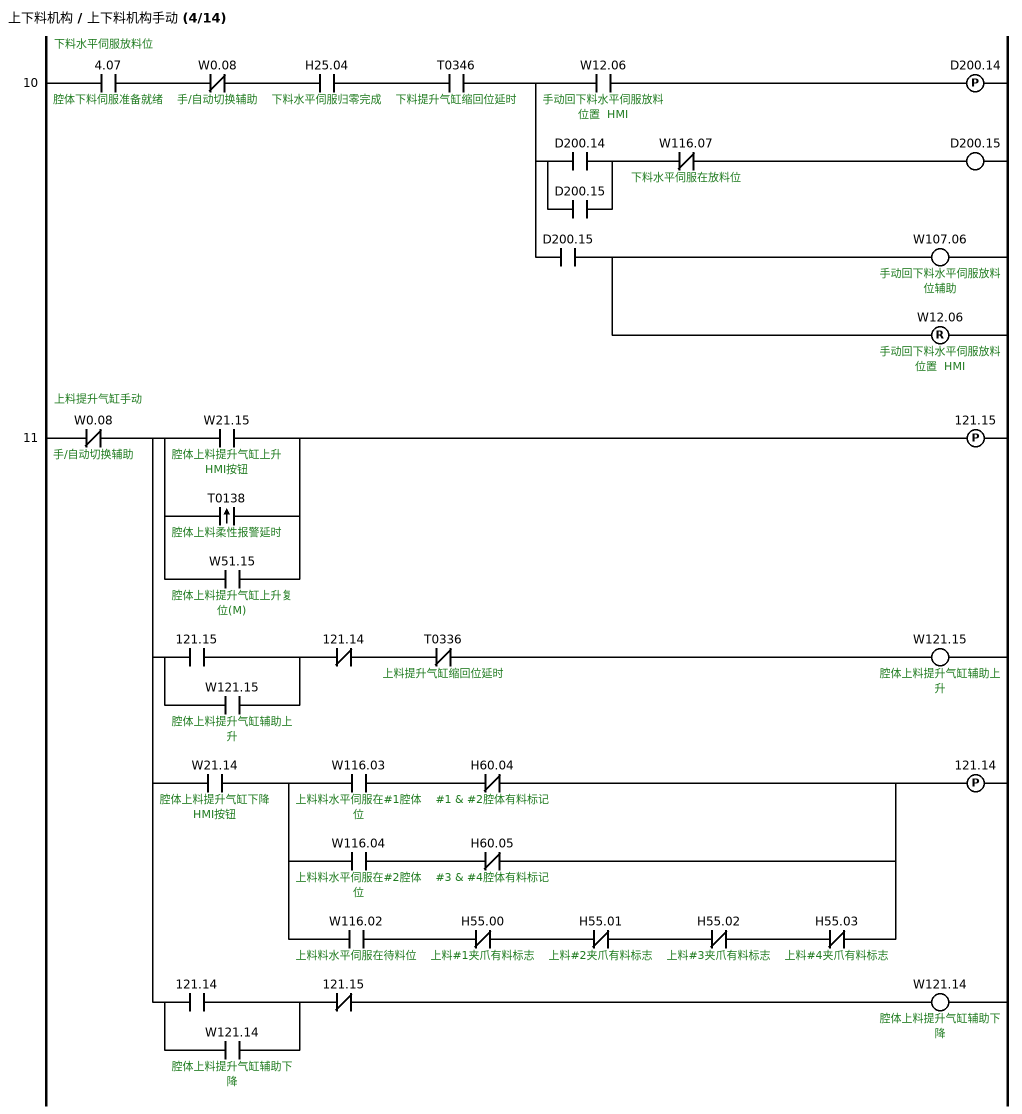
; [picture p192: 上下料机构 / 上下料机构手动, rungs 10-11]
; rung 10: 下料水平伺服放料位
LD 4.07  ; 腔体下料伺服准备就绪
ANDNOT W0.08  ; 手/自动切换辅助
AND H25.04  ; 下料水平伺服归零完成
AND T0346  ; 下料提升气缸缩回位延时
OUT TR0
AND W12.06  ; 手动回下料水平伺服放料位置  HMI
DIFU(013) D200.14
LD TR0
LD D200.14
OR D200.15
ANDLD
ANDNOT W116.07  ; 下料水平伺服在放料位
OUT D200.15
LD TR0
AND D200.15
OUT W107.06  ; 手动回下料水平伺服放料位辅助
RSET W12.06  ; 手动回下料水平伺服放料位置  HMI
; rung 11: 上料提升气缸手动
LDNOT W0.08  ; 手/自动切换辅助
OUT TR0
LD W21.15  ; 腔体上料提升气缸上升   HMI按钮
@OR T0138  ; 腔体上料柔性报警延时
OR W51.15  ; 腔体上料提升气缸上升复位(M)
ANDLD
DIFU(013) 121.15
LD TR0
LD 121.15
OR W121.15  ; 腔体上料提升气缸辅助上升
ANDLD
ANDNOT 121.14
ANDNOT T0336  ; 上料提升气缸缩回位延时
OUT W121.15  ; 腔体上料提升气缸辅助上升
LD TR0
AND W21.14  ; 腔体上料提升气缸下降   HMI按钮
LD W116.03  ; 上料料水平伺服在#1腔体位
ANDNOT H60.04  ; #1 & #2腔体有料标记
LD W116.04  ; 上料料水平伺服在#2腔体位
ANDNOT H60.05  ; #3 & #4腔体有料标记
ORLD
LD W116.02  ; 上料料水平伺服在待料位
ANDNOT H55.00  ; 上料#1夹爪有料标志
ANDNOT H55.01  ; 上料#2夹爪有料标志
ANDNOT H55.02  ; 上料#3夹爪有料标志
ANDNOT H55.03  ; 上料#4夹爪有料标志
ORLD
ANDLD
DIFU(013) 121.14
LD TR0
LD 121.14
OR W121.14  ; 腔体上料提升气缸辅助下降
ANDLD
ANDNOT 121.15
OUT W121.14  ; 腔体上料提升气缸辅助下降

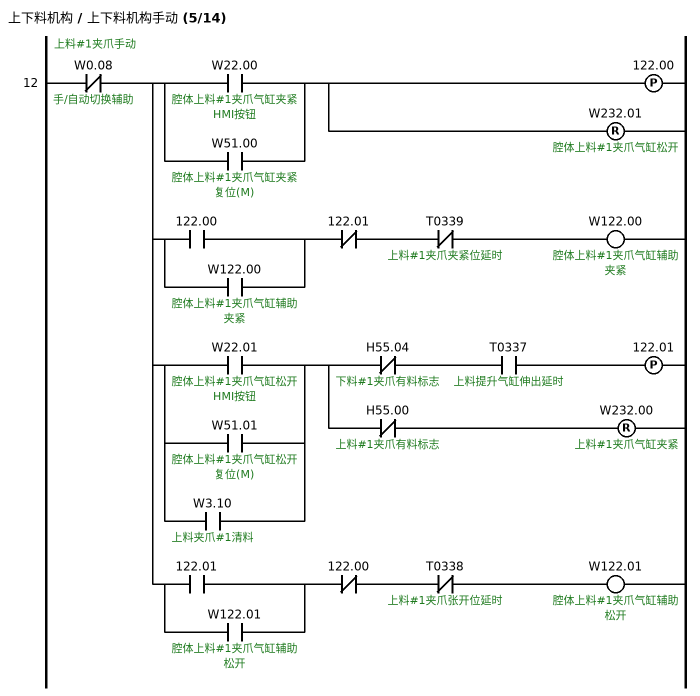
; rung 12: 上料#1夹爪手动
LDNOT W0.08  ; 手/自动切换辅助
OUT TR0
LD W22.00  ; 腔体上料#1夹爪气缸夹紧   HMI按钮
OR W51.00  ; 腔体上料#1夹爪气缸夹紧复位(M)
ANDLD
DIFU(013) 122.00
RSET W232.01  ; 腔体上料#1夹爪气缸松开
LD TR0
LD 122.00
OR W122.00  ; 腔体上料#1夹爪气缸辅助夹紧
ANDLD
ANDNOT 122.01
ANDNOT T0339  ; 上料#1夹爪夹紧位延时
OUT W122.00  ; 腔体上料#1夹爪气缸辅助夹紧
LD TR0
LD W22.01  ; 腔体上料#1夹爪气缸松开   HMI按钮
OR W51.01  ; 腔体上料#1夹爪气缸松开复位(M)
OR W3.10  ; 上料夹爪#1清料
ANDLD
OUT TR1
ANDNOT H55.04  ; 下料#1夹爪有料标志
AND T0337  ; 上料提升气缸伸出延时
DIFU(013) 122.01
LD TR1
ANDNOT H55.00  ; 上料#1夹爪有料标志
RSET W232.00  ; 上料#1夹爪气缸夹紧
LD TR0
LD 122.01
OR W122.01  ; 腔体上料#1夹爪气缸辅助松开
ANDLD
ANDNOT 122.00
ANDNOT T0338  ; 上料#1夹爪张开位延时
OUT W122.01  ; 腔体上料#1夹爪气缸辅助松开

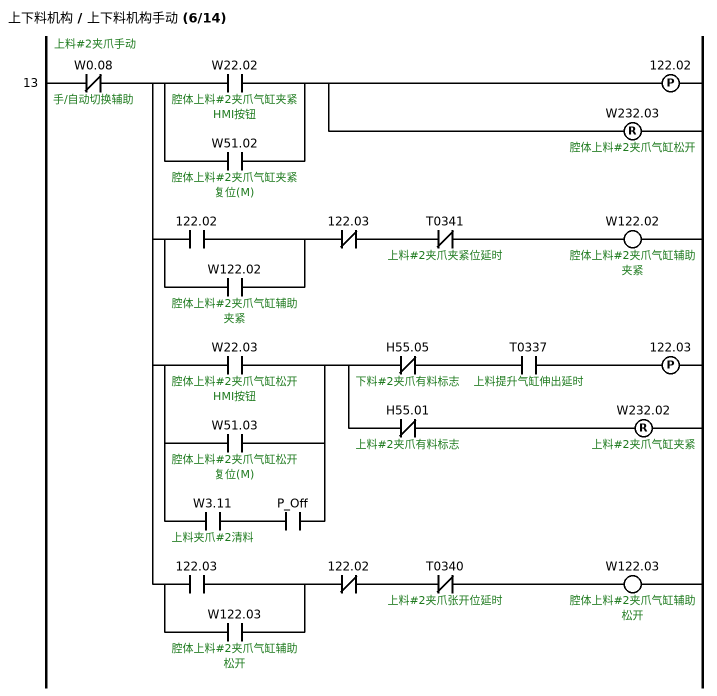
; rung 13: 上料#2夹爪手动
LDNOT W0.08  ; 手/自动切换辅助
OUT TR0
LD W22.02  ; 腔体上料#2夹爪气缸夹紧   HMI按钮
OR W51.02  ; 腔体上料#2夹爪气缸夹紧复位(M)
ANDLD
DIFU(013) 122.02
RSET W232.03  ; 腔体上料#2夹爪气缸松开
LD TR0
LD 122.02
OR W122.02  ; 腔体上料#2夹爪气缸辅助夹紧
ANDLD
ANDNOT 122.03
ANDNOT T0341  ; 上料#2夹爪夹紧位延时
OUT W122.02  ; 腔体上料#2夹爪气缸辅助夹紧
LD TR0
LD W22.03  ; 腔体上料#2夹爪气缸松开   HMI按钮
OR W51.03  ; 腔体上料#2夹爪气缸松开复位(M)
LD W3.11  ; 上料夹爪#2清料
AND P_Off
ORLD
ANDLD
OUT TR1
ANDNOT H55.05  ; 下料#2夹爪有料标志
AND T0337  ; 上料提升气缸伸出延时
DIFU(013) 122.03
LD TR1
ANDNOT H55.01  ; 上料#2夹爪有料标志
RSET W232.02  ; 上料#2夹爪气缸夹紧
LD TR0
LD 122.03
OR W122.03  ; 腔体上料#2夹爪气缸辅助松开
ANDLD
ANDNOT 122.02
ANDNOT T0340  ; 上料#2夹爪张开位延时
OUT W122.03  ; 腔体上料#2夹爪气缸辅助松开

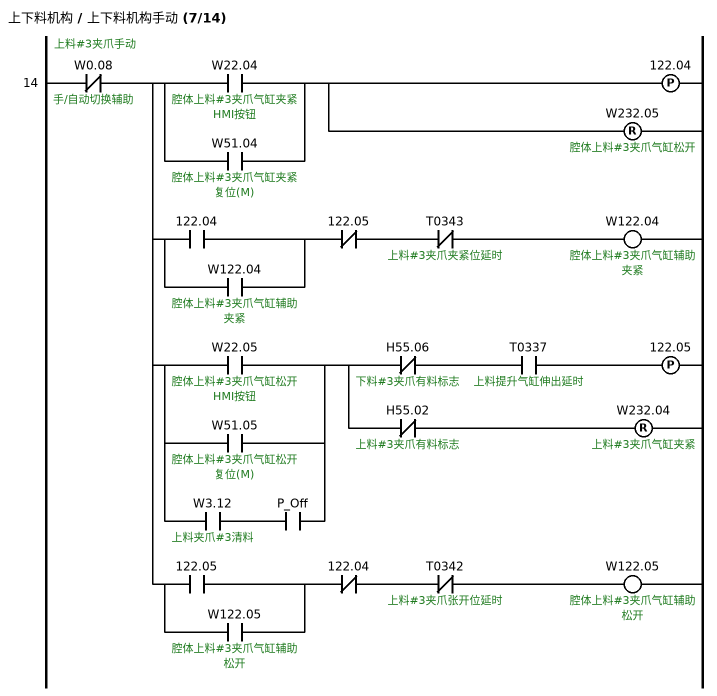
; rung 14: 上料#3夹爪手动
LDNOT W0.08  ; 手/自动切换辅助
OUT TR0
LD W22.04  ; 腔体上料#3夹爪气缸夹紧   HMI按钮
OR W51.04  ; 腔体上料#3夹爪气缸夹紧复位(M)
ANDLD
DIFU(013) 122.04
RSET W232.05  ; 腔体上料#3夹爪气缸松开
LD TR0
LD 122.04
OR W122.04  ; 腔体上料#3夹爪气缸辅助夹紧
ANDLD
ANDNOT 122.05
ANDNOT T0343  ; 上料#3夹爪夹紧位延时
OUT W122.04  ; 腔体上料#3夹爪气缸辅助夹紧
LD TR0
LD W22.05  ; 腔体上料#3夹爪气缸松开   HMI按钮
OR W51.05  ; 腔体上料#3夹爪气缸松开复位(M)
LD W3.12  ; 上料夹爪#3清料
AND P_Off
ORLD
ANDLD
OUT TR1
ANDNOT H55.06  ; 下料#3夹爪有料标志
AND T0337  ; 上料提升气缸伸出延时
DIFU(013) 122.05
LD TR1
ANDNOT H55.02  ; 上料#3夹爪有料标志
RSET W232.04  ; 上料#3夹爪气缸夹紧
LD TR0
LD 122.05
OR W122.05  ; 腔体上料#3夹爪气缸辅助松开
ANDLD
ANDNOT 122.04
ANDNOT T0342  ; 上料#3夹爪张开位延时
OUT W122.05  ; 腔体上料#3夹爪气缸辅助松开

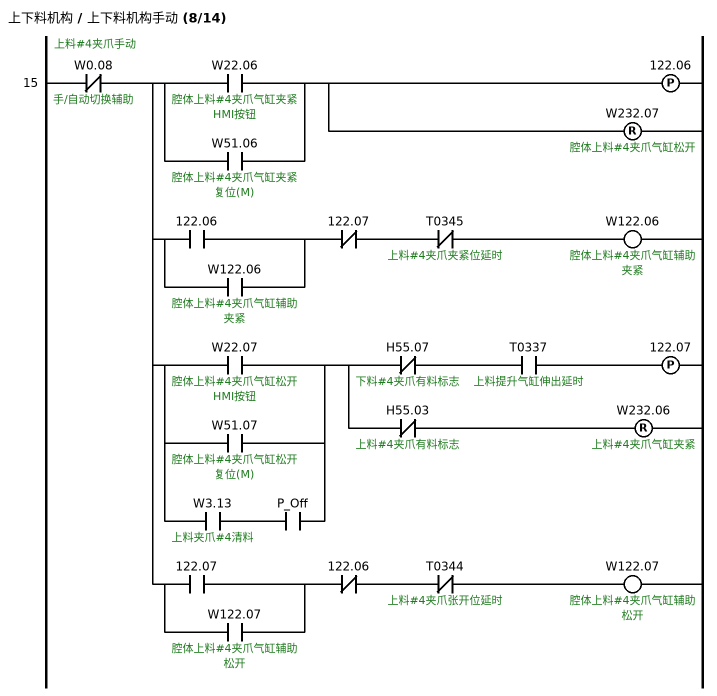
; rung 15: 上料#4夹爪手动
LDNOT W0.08  ; 手/自动切换辅助
OUT TR0
LD W22.06  ; 腔体上料#4夹爪气缸夹紧   HMI按钮
OR W51.06  ; 腔体上料#4夹爪气缸夹紧复位(M)
ANDLD
DIFU(013) 122.06
RSET W232.07  ; 腔体上料#4夹爪气缸松开
LD TR0
LD 122.06
OR W122.06  ; 腔体上料#4夹爪气缸辅助夹紧
ANDLD
ANDNOT 122.07
ANDNOT T0345  ; 上料#4夹爪夹紧位延时
OUT W122.06  ; 腔体上料#4夹爪气缸辅助夹紧
LD TR0
LD W22.07  ; 腔体上料#4夹爪气缸松开   HMI按钮
OR W51.07  ; 腔体上料#4夹爪气缸松开复位(M)
LD W3.13  ; 上料夹爪#4清料
AND P_Off
ORLD
ANDLD
OUT TR1
ANDNOT H55.07  ; 下料#4夹爪有料标志
AND T0337  ; 上料提升气缸伸出延时
DIFU(013) 122.07
LD TR1
ANDNOT H55.03  ; 上料#4夹爪有料标志
RSET W232.06  ; 上料#4夹爪气缸夹紧
LD TR0
LD 122.07
OR W122.07  ; 腔体上料#4夹爪气缸辅助松开
ANDLD
ANDNOT 122.06
ANDNOT T0344  ; 上料#4夹爪张开位延时
OUT W122.07  ; 腔体上料#4夹爪气缸辅助松开

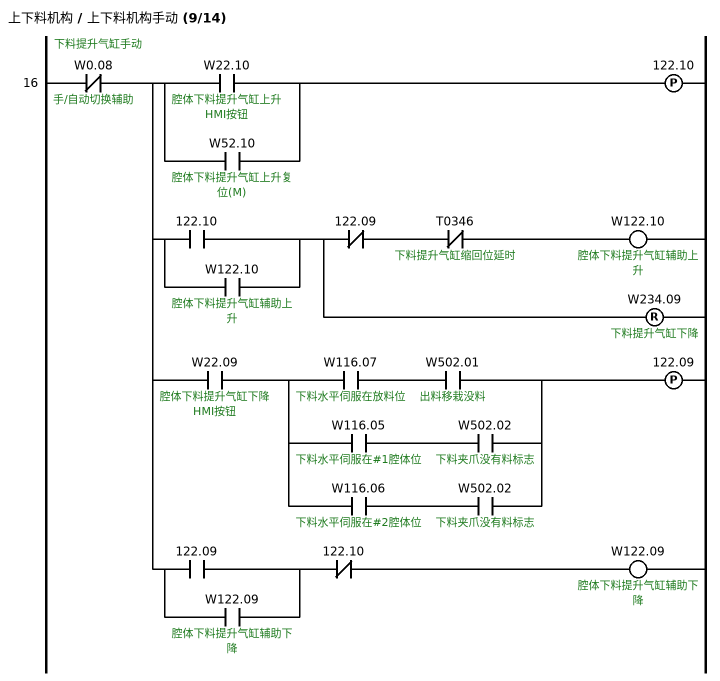
; rung 16: 下料提升气缸手动
LDNOT W0.08  ; 手/自动切换辅助
OUT TR0
LD W22.10  ; 腔体下料提升气缸上升   HMI按钮
OR W52.10  ; 腔体下料提升气缸上升复位(M)
ANDLD
DIFU(013) 122.10
LD TR0
LD 122.10
OR W122.10  ; 腔体下料提升气缸辅助上升
ANDLD
OUT TR1
ANDNOT 122.09
ANDNOT T0346  ; 下料提升气缸缩回位延时
OUT W122.10  ; 腔体下料提升气缸辅助上升
LD TR1
RSET W234.09  ; 下料提升气缸下降
LD TR0
AND W22.09  ; 腔体下料提升气缸下降   HMI按钮
LD W116.07  ; 下料水平伺服在放料位
AND W502.01  ; 出料移栽没料
LD W116.05  ; 下料水平伺服在#1腔体位
AND W502.02  ; 下料夹爪没有料标志
ORLD
LD W116.06  ; 下料水平伺服在#2腔体位
AND W502.02  ; 下料夹爪没有料标志
ORLD
ANDLD
DIFU(013) 122.09
LD TR0
LD 122.09
OR W122.09  ; 腔体下料提升气缸辅助下降
ANDLD
ANDNOT 122.10
OUT W122.09  ; 腔体下料提升气缸辅助下降

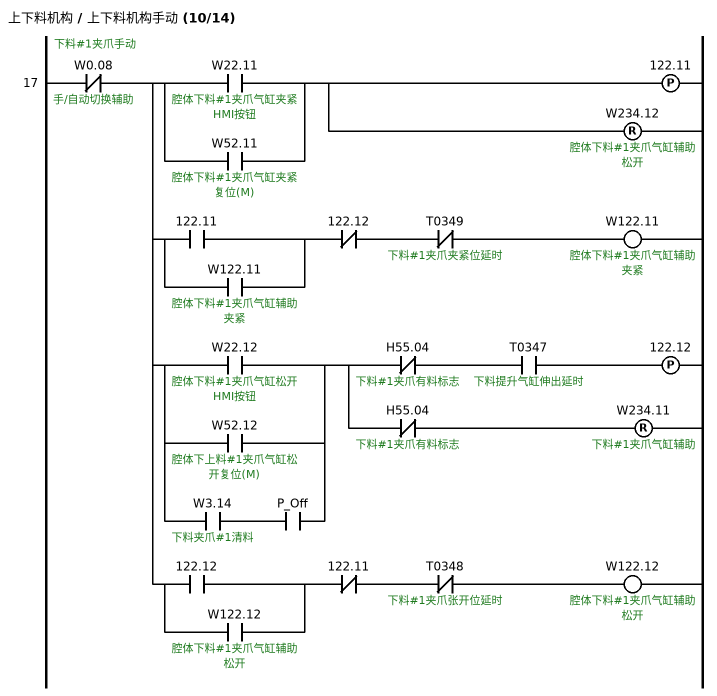
; rung 17: 下料#1夹爪手动
LDNOT W0.08  ; 手/自动切换辅助
OUT TR0
LD W22.11  ; 腔体下料#1夹爪气缸夹紧   HMI按钮
OR W52.11  ; 腔体下料#1夹爪气缸夹紧复位(M)
ANDLD
DIFU(013) 122.11
RSET W234.12  ; 腔体下料#1夹爪气缸辅助松开
LD TR0
LD 122.11
OR W122.11  ; 腔体下料#1夹爪气缸辅助夹紧
ANDLD
ANDNOT 122.12
ANDNOT T0349  ; 下料#1夹爪夹紧位延时
OUT W122.11  ; 腔体下料#1夹爪气缸辅助夹紧
LD TR0
LD W22.12  ; 腔体下料#1夹爪气缸松开   HMI按钮
OR W52.12  ; 腔体下上料#1夹爪气缸松开复位(M)
LD W3.14  ; 下料夹爪#1清料
AND P_Off
ORLD
ANDLD
OUT TR1
ANDNOT H55.04  ; 下料#1夹爪有料标志
AND T0347  ; 下料提升气缸伸出延时
DIFU(013) 122.12
LD TR1
ANDNOT H55.04  ; 下料#1夹爪有料标志
RSET W234.11  ; 下料#1夹爪气缸辅助
LD TR0
LD 122.12
OR W122.12  ; 腔体下料#1夹爪气缸辅助松开
ANDLD
ANDNOT 122.11
ANDNOT T0348  ; 下料#1夹爪张开位延时
OUT W122.12  ; 腔体下料#1夹爪气缸辅助松开

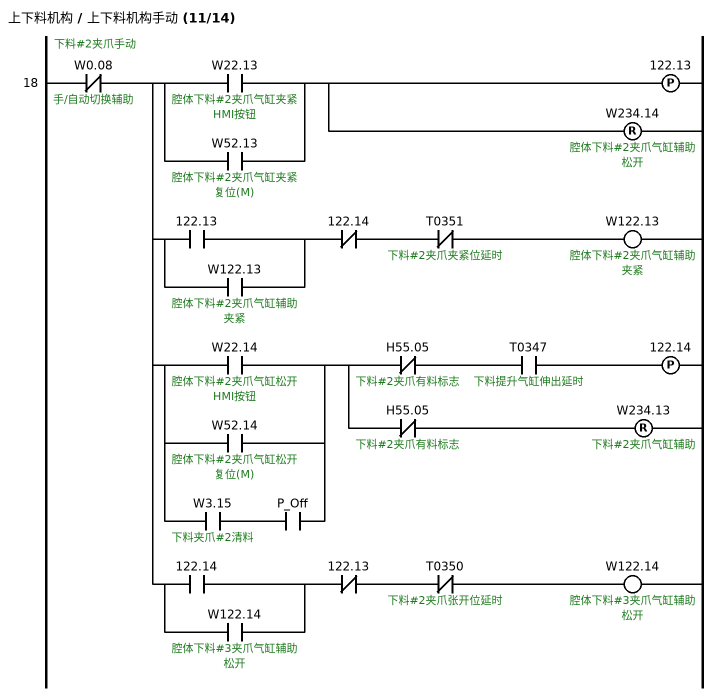
; rung 18: 下料#2夹爪手动
LDNOT W0.08  ; 手/自动切换辅助
OUT TR0
LD W22.13  ; 腔体下料#2夹爪气缸夹紧   HMI按钮
OR W52.13  ; 腔体下料#2夹爪气缸夹紧复位(M)
ANDLD
DIFU(013) 122.13
RSET W234.14  ; 腔体下料#2夹爪气缸辅助松开
LD TR0
LD 122.13
OR W122.13  ; 腔体下料#2夹爪气缸辅助夹紧
ANDLD
ANDNOT 122.14
ANDNOT T0351  ; 下料#2夹爪夹紧位延时
OUT W122.13  ; 腔体下料#2夹爪气缸辅助夹紧
LD TR0
LD W22.14  ; 腔体下料#2夹爪气缸松开   HMI按钮
OR W52.14  ; 腔体下料#2夹爪气缸松开复位(M)
LD W3.15  ; 下料夹爪#2清料
AND P_Off
ORLD
ANDLD
OUT TR1
ANDNOT H55.05  ; 下料#2夹爪有料标志
AND T0347  ; 下料提升气缸伸出延时
DIFU(013) 122.14
LD TR1
ANDNOT H55.05  ; 下料#2夹爪有料标志
RSET W234.13  ; 下料#2夹爪气缸辅助
LD TR0
LD 122.14
OR W122.14  ; 腔体下料#3夹爪气缸辅助松开
ANDLD
ANDNOT 122.13
ANDNOT T0350  ; 下料#2夹爪张开位延时
OUT W122.14  ; 腔体下料#3夹爪气缸辅助松开

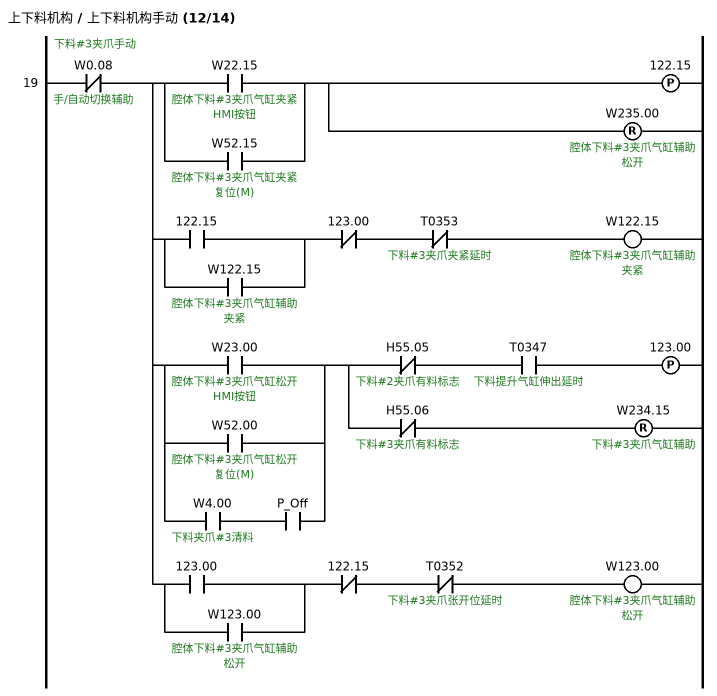
; rung 19: 下料#3夹爪手动
LDNOT W0.08  ; 手/自动切换辅助
OUT TR0
LD W22.15  ; 腔体下料#3夹爪气缸夹紧   HMI按钮
OR W52.15  ; 腔体下料#3夹爪气缸夹紧复位(M)
ANDLD
DIFU(013) 122.15
RSET W235.00  ; 腔体下料#3夹爪气缸辅助松开
LD TR0
LD 122.15
OR W122.15  ; 腔体下料#3夹爪气缸辅助夹紧
ANDLD
ANDNOT 123.00
ANDNOT T0353  ; 下料#3夹爪夹紧延时
OUT W122.15  ; 腔体下料#3夹爪气缸辅助夹紧
LD TR0
LD W23.00  ; 腔体下料#3夹爪气缸松开   HMI按钮
OR W52.00  ; 腔体下料#3夹爪气缸松开复位(M)
LD W4.00  ; 下料夹爪#3清料
AND P_Off
ORLD
ANDLD
OUT TR1
ANDNOT H55.05  ; 下料#2夹爪有料标志
AND T0347  ; 下料提升气缸伸出延时
DIFU(013) 123.00
LD TR1
ANDNOT H55.06  ; 下料#3夹爪有料标志
RSET W234.15  ; 下料#3夹爪气缸辅助
LD TR0
LD 123.00
OR W123.00  ; 腔体下料#3夹爪气缸辅助松开
ANDLD
ANDNOT 122.15
ANDNOT T0352  ; 下料#3夹爪张开位延时
OUT W123.00  ; 腔体下料#3夹爪气缸辅助松开

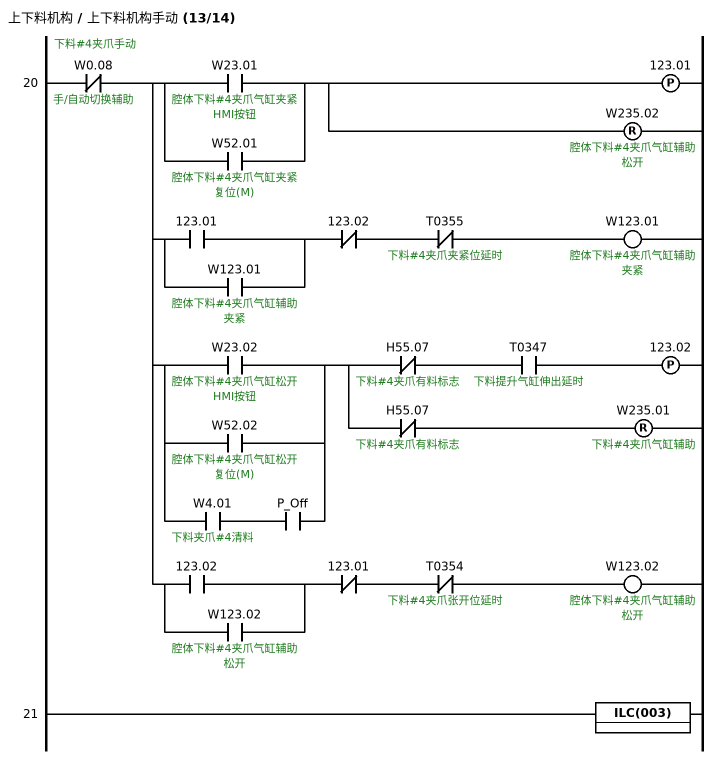
; rung 20: 下料#4夹爪手动
LDNOT W0.08  ; 手/自动切换辅助
OUT TR0
LD W23.01  ; 腔体下料#4夹爪气缸夹紧   HMI按钮
OR W52.01  ; 腔体下料#4夹爪气缸夹紧复位(M)
ANDLD
DIFU(013) 123.01
RSET W235.02  ; 腔体下料#4夹爪气缸辅助松开
LD TR0
LD 123.01
OR W123.01  ; 腔体下料#4夹爪气缸辅助夹紧
ANDLD
ANDNOT 123.02
ANDNOT T0355  ; 下料#4夹爪夹紧位延时
OUT W123.01  ; 腔体下料#4夹爪气缸辅助夹紧
LD TR0
LD W23.02  ; 腔体下料#4夹爪气缸松开   HMI按钮
OR W52.02  ; 腔体下料#4夹爪气缸松开复位(M)
LD W4.01  ; 下料夹爪#4清料
AND P_Off
ORLD
ANDLD
OUT TR1
ANDNOT H55.07  ; 下料#4夹爪有料标志
AND T0347  ; 下料提升气缸伸出延时
DIFU(013) 123.02
LD TR1
ANDNOT H55.07  ; 下料#4夹爪有料标志
RSET W235.01  ; 下料#4夹爪气缸辅助
LD TR0
LD 123.02
OR W123.02  ; 腔体下料#4夹爪气缸辅助松开
ANDLD
ANDNOT 123.01
ANDNOT T0354  ; 下料#4夹爪张开位延时
OUT W123.02  ; 腔体下料#4夹爪气缸辅助松开
; rung 21
ILC(003)

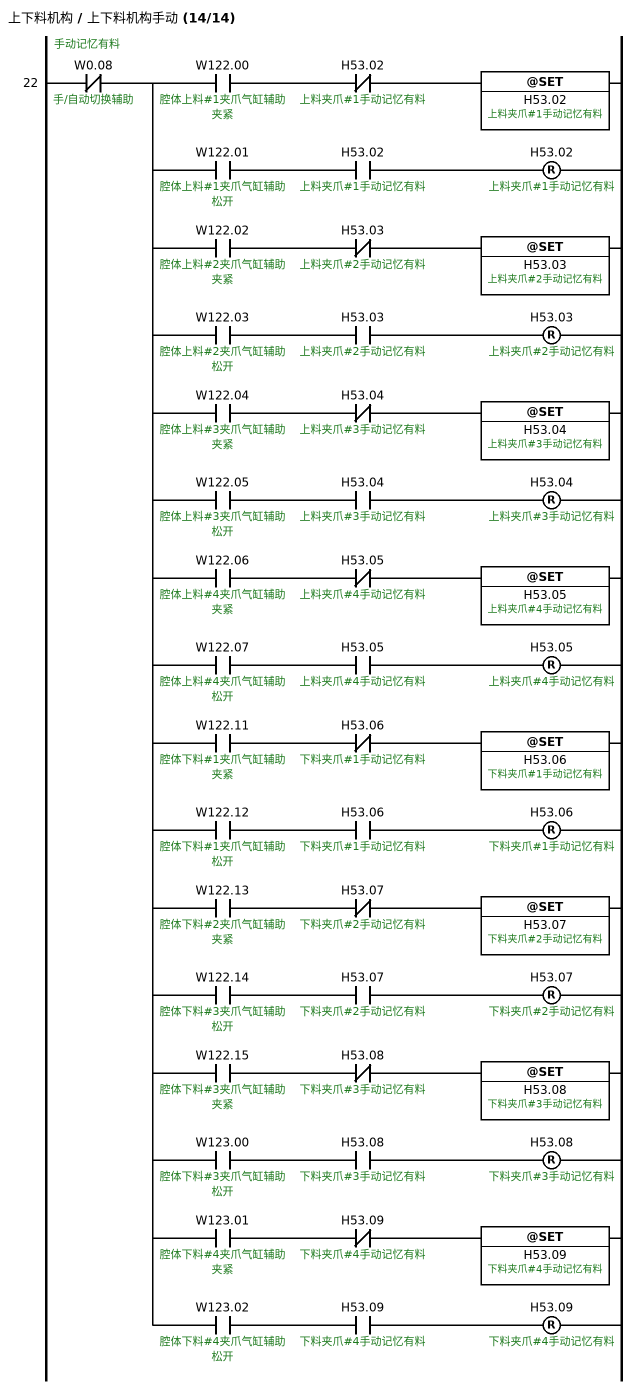
; rung 22: 手动记忆有料
LDNOT W0.08  ; 手/自动切换辅助
OUT TR0
AND W122.00  ; 腔体上料#1夹爪气缸辅助夹紧
ANDNOT H53.02  ; 上料夹爪#1手动记忆有料
@SET H53.02  ; 上料夹爪#1手动记忆有料
LD TR0
AND W122.01  ; 腔体上料#1夹爪气缸辅助松开
AND H53.02  ; 上料夹爪#1手动记忆有料
RSET H53.02  ; 上料夹爪#1手动记忆有料
LD TR0
AND W122.02  ; 腔体上料#2夹爪气缸辅助夹紧
ANDNOT H53.03  ; 上料夹爪#2手动记忆有料
@SET H53.03  ; 上料夹爪#2手动记忆有料
LD TR0
AND W122.03  ; 腔体上料#2夹爪气缸辅助松开
AND H53.03  ; 上料夹爪#2手动记忆有料
RSET H53.03  ; 上料夹爪#2手动记忆有料
LD TR0
AND W122.04  ; 腔体上料#3夹爪气缸辅助夹紧
ANDNOT H53.04  ; 上料夹爪#3手动记忆有料
@SET H53.04  ; 上料夹爪#3手动记忆有料
LD TR0
AND W122.05  ; 腔体上料#3夹爪气缸辅助松开
AND H53.04  ; 上料夹爪#3手动记忆有料
RSET H53.04  ; 上料夹爪#3手动记忆有料
LD TR0
AND W122.06  ; 腔体上料#4夹爪气缸辅助夹紧
ANDNOT H53.05  ; 上料夹爪#4手动记忆有料
@SET H53.05  ; 上料夹爪#4手动记忆有料
LD TR0
AND W122.07  ; 腔体上料#4夹爪气缸辅助松开
AND H53.05  ; 上料夹爪#4手动记忆有料
RSET H53.05  ; 上料夹爪#4手动记忆有料
LD TR0
AND W122.11  ; 腔体下料#1夹爪气缸辅助夹紧
ANDNOT H53.06  ; 下料夹爪#1手动记忆有料
@SET H53.06  ; 下料夹爪#1手动记忆有料
LD TR0
AND W122.12  ; 腔体下料#1夹爪气缸辅助松开
AND H53.06  ; 下料夹爪#1手动记忆有料
RSET H53.06  ; 下料夹爪#1手动记忆有料
LD TR0
AND W122.13  ; 腔体下料#2夹爪气缸辅助夹紧
ANDNOT H53.07  ; 下料夹爪#2手动记忆有料
@SET H53.07  ; 下料夹爪#2手动记忆有料
LD TR0
AND W122.14  ; 腔体下料#3夹爪气缸辅助松开
AND H53.07  ; 下料夹爪#2手动记忆有料
RSET H53.07  ; 下料夹爪#2手动记忆有料
LD TR0
AND W122.15  ; 腔体下料#3夹爪气缸辅助夹紧
ANDNOT H53.08  ; 下料夹爪#3手动记忆有料
@SET H53.08  ; 下料夹爪#3手动记忆有料
LD TR0
AND W123.00  ; 腔体下料#3夹爪气缸辅助松开
AND H53.08  ; 下料夹爪#3手动记忆有料
RSET H53.08  ; 下料夹爪#3手动记忆有料
LD TR0
AND W123.01  ; 腔体下料#4夹爪气缸辅助夹紧
ANDNOT H53.09  ; 下料夹爪#4手动记忆有料
@SET H53.09  ; 下料夹爪#4手动记忆有料
LD TR0
AND W123.02  ; 腔体下料#4夹爪气缸辅助松开
AND H53.09  ; 下料夹爪#4手动记忆有料
RSET H53.09  ; 下料夹爪#4手动记忆有料

### Section 上下料机构输出

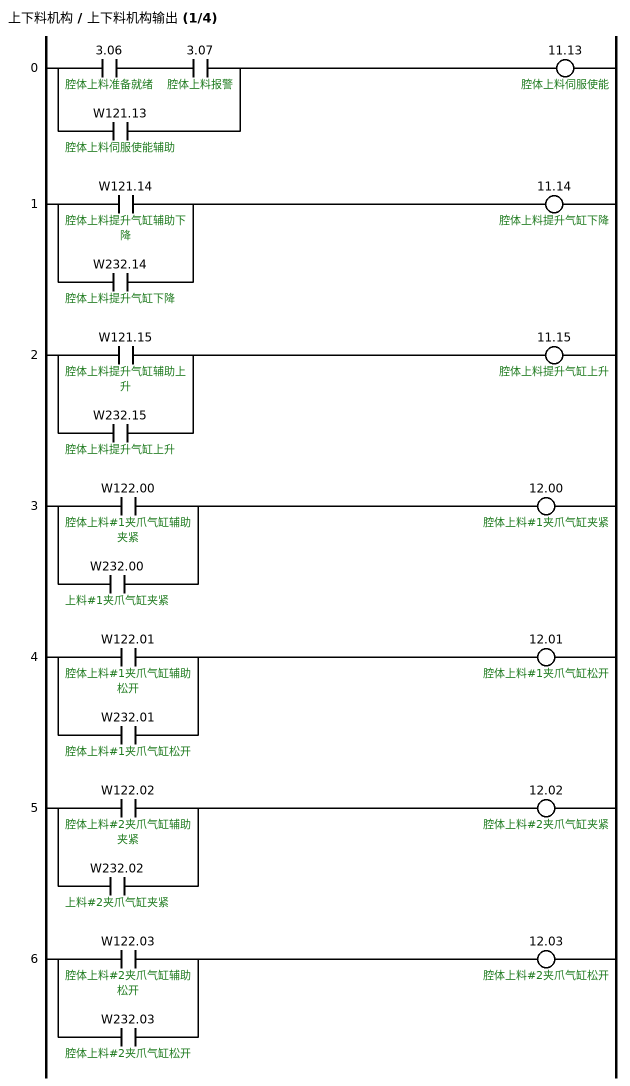
; rung 0
LD 3.06  ; 腔体上料准备就绪
AND 3.07  ; 腔体上料报警
OR W121.13  ; 腔体上料伺服使能辅助
OUT 11.13  ; 腔体上料伺服使能
; rung 1
LD W121.14  ; 腔体上料提升气缸辅助下降
OR W232.14  ; 腔体上料提升气缸下降
OUT 11.14  ; 腔体上料提升气缸下降
; rung 2
LD W121.15  ; 腔体上料提升气缸辅助上升
OR W232.15  ; 腔体上料提升气缸上升
OUT 11.15  ; 腔体上料提升气缸上升
; rung 3
LD W122.00  ; 腔体上料#1夹爪气缸辅助夹紧
OR W232.00  ; 上料#1夹爪气缸夹紧
OUT 12.00  ; 腔体上料#1夹爪气缸夹紧
; rung 4
LD W122.01  ; 腔体上料#1夹爪气缸辅助松开
OR W232.01  ; 腔体上料#1夹爪气缸松开
OUT 12.01  ; 腔体上料#1夹爪气缸松开
; rung 5
LD W122.02  ; 腔体上料#2夹爪气缸辅助夹紧
OR W232.02  ; 上料#2夹爪气缸夹紧
OUT 12.02  ; 腔体上料#2夹爪气缸夹紧
; rung 6
LD W122.03  ; 腔体上料#2夹爪气缸辅助松开
OR W232.03  ; 腔体上料#2夹爪气缸松开
OUT 12.03  ; 腔体上料#2夹爪气缸松开

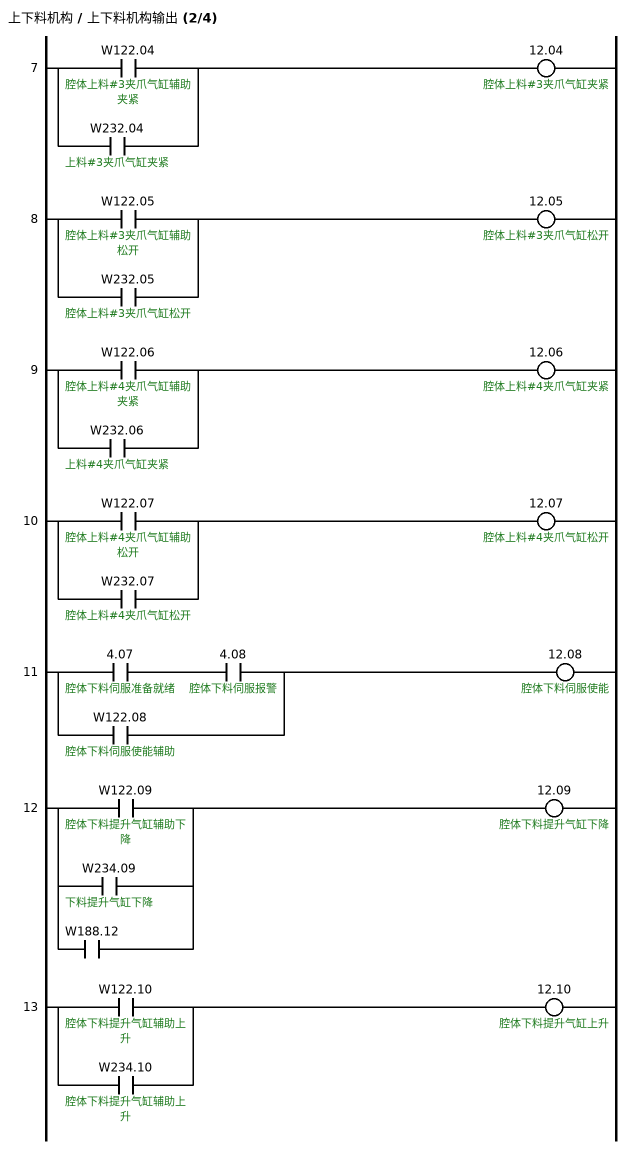
; rung 7
LD W122.04  ; 腔体上料#3夹爪气缸辅助夹紧
OR W232.04  ; 上料#3夹爪气缸夹紧
OUT 12.04  ; 腔体上料#3夹爪气缸夹紧
; rung 8
LD W122.05  ; 腔体上料#3夹爪气缸辅助松开
OR W232.05  ; 腔体上料#3夹爪气缸松开
OUT 12.05  ; 腔体上料#3夹爪气缸松开
; rung 9
LD W122.06  ; 腔体上料#4夹爪气缸辅助夹紧
OR W232.06  ; 上料#4夹爪气缸夹紧
OUT 12.06  ; 腔体上料#4夹爪气缸夹紧
; rung 10
LD W122.07  ; 腔体上料#4夹爪气缸辅助松开
OR W232.07  ; 腔体上料#4夹爪气缸松开
OUT 12.07  ; 腔体上料#4夹爪气缸松开
; rung 11
LD 4.07  ; 腔体下料伺服准备就绪
AND 4.08  ; 腔体下料伺服报警
OR W122.08  ; 腔体下料伺服使能辅助
OUT 12.08  ; 腔体下料伺服使能
; rung 12
LD W122.09  ; 腔体下料提升气缸辅助下降
OR W234.09  ; 下料提升气缸下降
OR W188.12
OUT 12.09  ; 腔体下料提升气缸下降
; rung 13
LD W122.10  ; 腔体下料提升气缸辅助上升
OR W234.10  ; 腔体下料提升气缸辅助上升
OUT 12.10  ; 腔体下料提升气缸上升

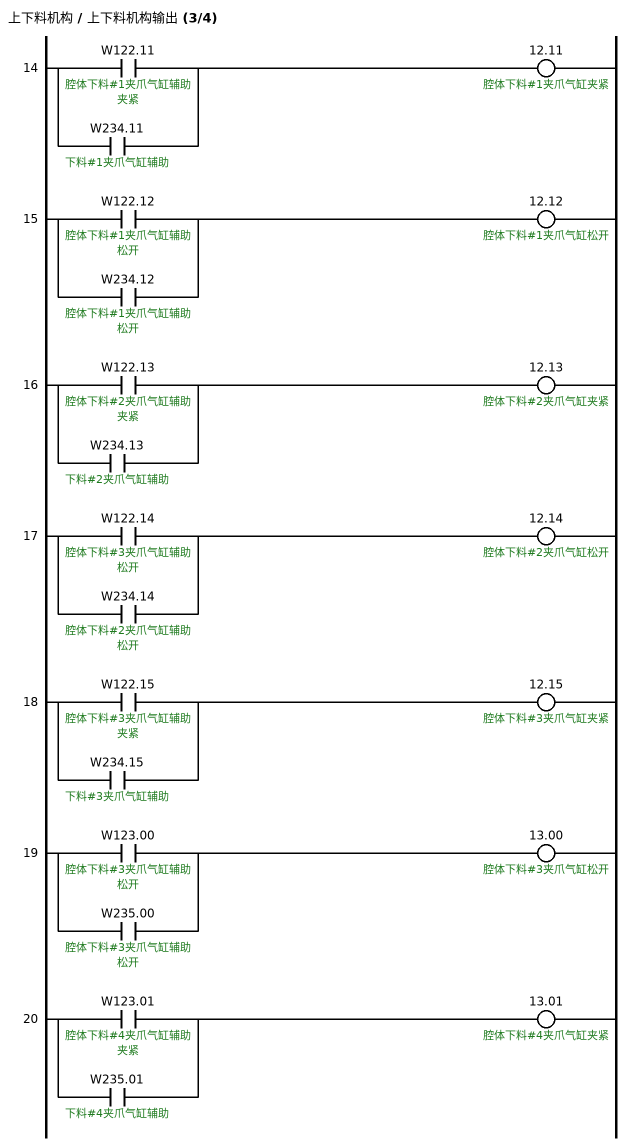
; rung 14
LD W122.11  ; 腔体下料#1夹爪气缸辅助夹紧
OR W234.11  ; 下料#1夹爪气缸辅助
OUT 12.11  ; 腔体下料#1夹爪气缸夹紧
; rung 15
LD W122.12  ; 腔体下料#1夹爪气缸辅助松开
OR W234.12  ; 腔体下料#1夹爪气缸辅助松开
OUT 12.12  ; 腔体下料#1夹爪气缸松开
; rung 16
LD W122.13  ; 腔体下料#2夹爪气缸辅助夹紧
OR W234.13  ; 下料#2夹爪气缸辅助
OUT 12.13  ; 腔体下料#2夹爪气缸夹紧
; rung 17
LD W122.14  ; 腔体下料#3夹爪气缸辅助松开
OR W234.14  ; 腔体下料#2夹爪气缸辅助松开
OUT 12.14  ; 腔体下料#2夹爪气缸松开
; rung 18
LD W122.15  ; 腔体下料#3夹爪气缸辅助夹紧
OR W234.15  ; 下料#3夹爪气缸辅助
OUT 12.15  ; 腔体下料#3夹爪气缸夹紧
; rung 19
LD W123.00  ; 腔体下料#3夹爪气缸辅助松开
OR W235.00  ; 腔体下料#3夹爪气缸辅助松开
OUT 13.00  ; 腔体下料#3夹爪气缸松开
; rung 20
LD W123.01  ; 腔体下料#4夹爪气缸辅助夹紧
OR W235.01  ; 下料#4夹爪气缸辅助
OUT 13.01  ; 腔体下料#4夹爪气缸夹紧

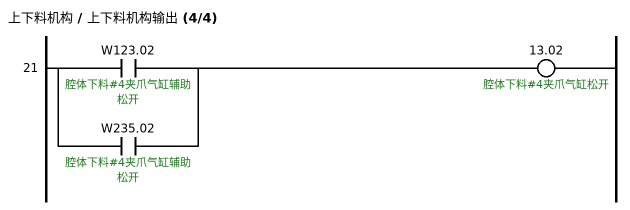
; rung 21
LD W123.02  ; 腔体下料#4夹爪气缸辅助松开
OR W235.02  ; 腔体下料#4夹爪气缸辅助松开
OUT 13.02  ; 腔体下料#4夹爪气缸松开

### Section 安全限制条件

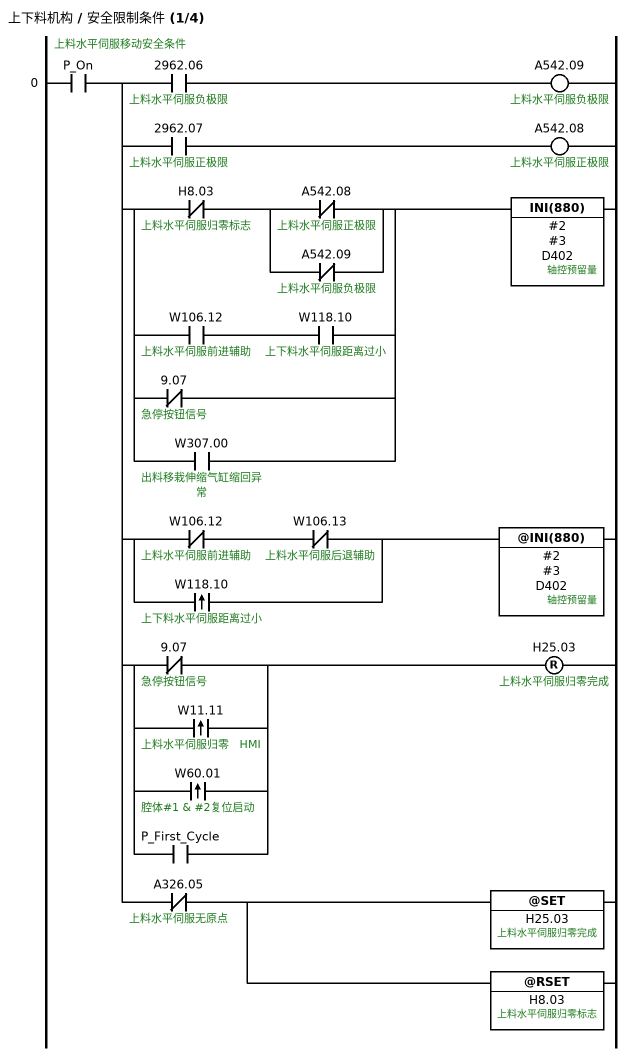
; rung 0: 上料水平伺服移动安全条件
LD P_On
OUT TR0
AND 2962.06  ; 上料水平伺服负极限
OUT A542.09  ; 上料水平伺服负极限
LD TR0
AND 2962.07  ; 上料水平伺服正极限
OUT A542.08  ; 上料水平伺服正极限
LD TR0
LDNOT H8.03  ; 上料水平伺服归零标志
LDNOT A542.08  ; 上料水平伺服正极限
ORNOT A542.09  ; 上料水平伺服负极限
ANDLD
LD W106.12  ; 上料水平伺服前进辅助
AND W118.10  ; 上下料水平伺服距离过小
ORLD
ORNOT 9.07  ; 急停按钮信号
OR W307.00  ; 出料移栽伸缩气缸缩回异常
ANDLD
INI(880) #2 #3 D402  ; 轴控预留量
LD TR0
LDNOT W106.12  ; 上料水平伺服前进辅助
ANDNOT W106.13  ; 上料水平伺服后退辅助
@OR W118.10  ; 上下料水平伺服距离过小
ANDLD
@INI(880) #2 #3 D402  ; 轴控预留量
LD TR0
LDNOT 9.07  ; 急停按钮信号
@OR W11.11  ; 上料水平伺服归零   HMI
@OR W60.01  ; 腔体#1 & #2复位启动
OR P_First_Cycle
ANDLD
RSET H25.03  ; 上料水平伺服归零完成
LD TR0
ANDNOT A326.05  ; 上料水平伺服无原点
@SET H25.03  ; 上料水平伺服归零完成
@RSET H8.03  ; 上料水平伺服归零标志

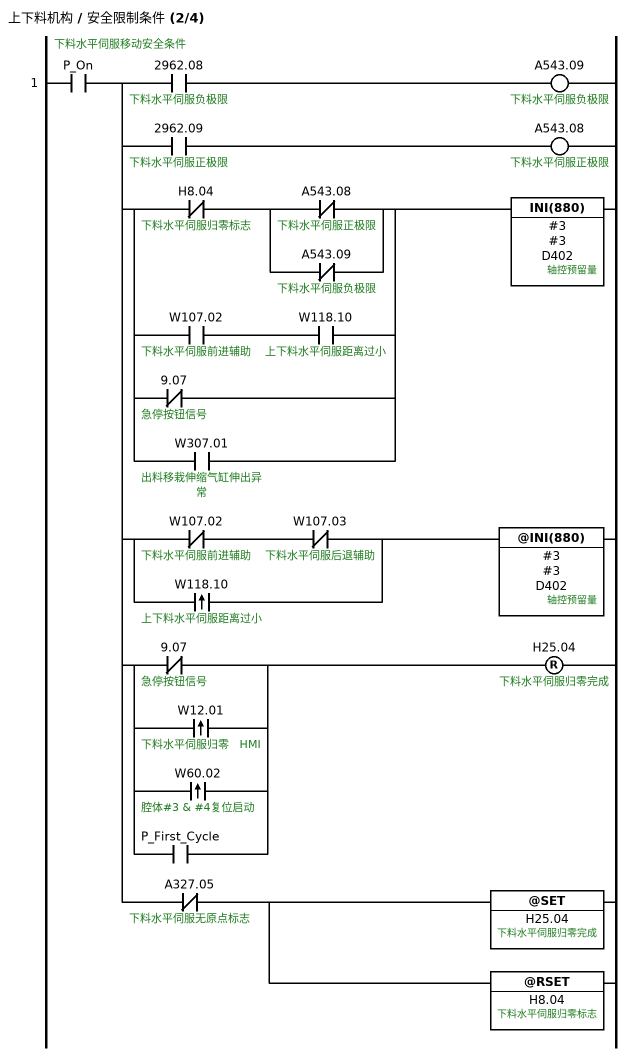
; rung 1: 下料水平伺服移动安全条件
LD P_On
OUT TR0
AND 2962.08  ; 下料水平伺服负极限
OUT A543.09  ; 下料水平伺服负极限
LD TR0
AND 2962.09  ; 下料水平伺服正极限
OUT A543.08  ; 下料水平伺服正极限
LD TR0
LDNOT H8.04  ; 下料水平伺服归零标志
LDNOT A543.08  ; 下料水平伺服正极限
ORNOT A543.09  ; 下料水平伺服负极限
ANDLD
LD W107.02  ; 下料水平伺服前进辅助
AND W118.10  ; 上下料水平伺服距离过小
ORLD
ORNOT 9.07  ; 急停按钮信号
OR W307.01  ; 出料移栽伸缩气缸伸出异常
ANDLD
INI(880) #3 #3 D402  ; 轴控预留量
LD TR0
LDNOT W107.02  ; 下料水平伺服前进辅助
ANDNOT W107.03  ; 下料水平伺服后退辅助
@OR W118.10  ; 上下料水平伺服距离过小
ANDLD
@INI(880) #3 #3 D402  ; 轴控预留量
LD TR0
LDNOT 9.07  ; 急停按钮信号
@OR W12.01  ; 下料水平伺服归零   HMI
@OR W60.02  ; 腔体#3 & #4复位启动
OR P_First_Cycle
ANDLD
RSET H25.04  ; 下料水平伺服归零完成
LD TR0
ANDNOT A327.05  ; 下料水平伺服无原点标志
@SET H25.04  ; 下料水平伺服归零完成
@RSET H8.04  ; 下料水平伺服归零标志

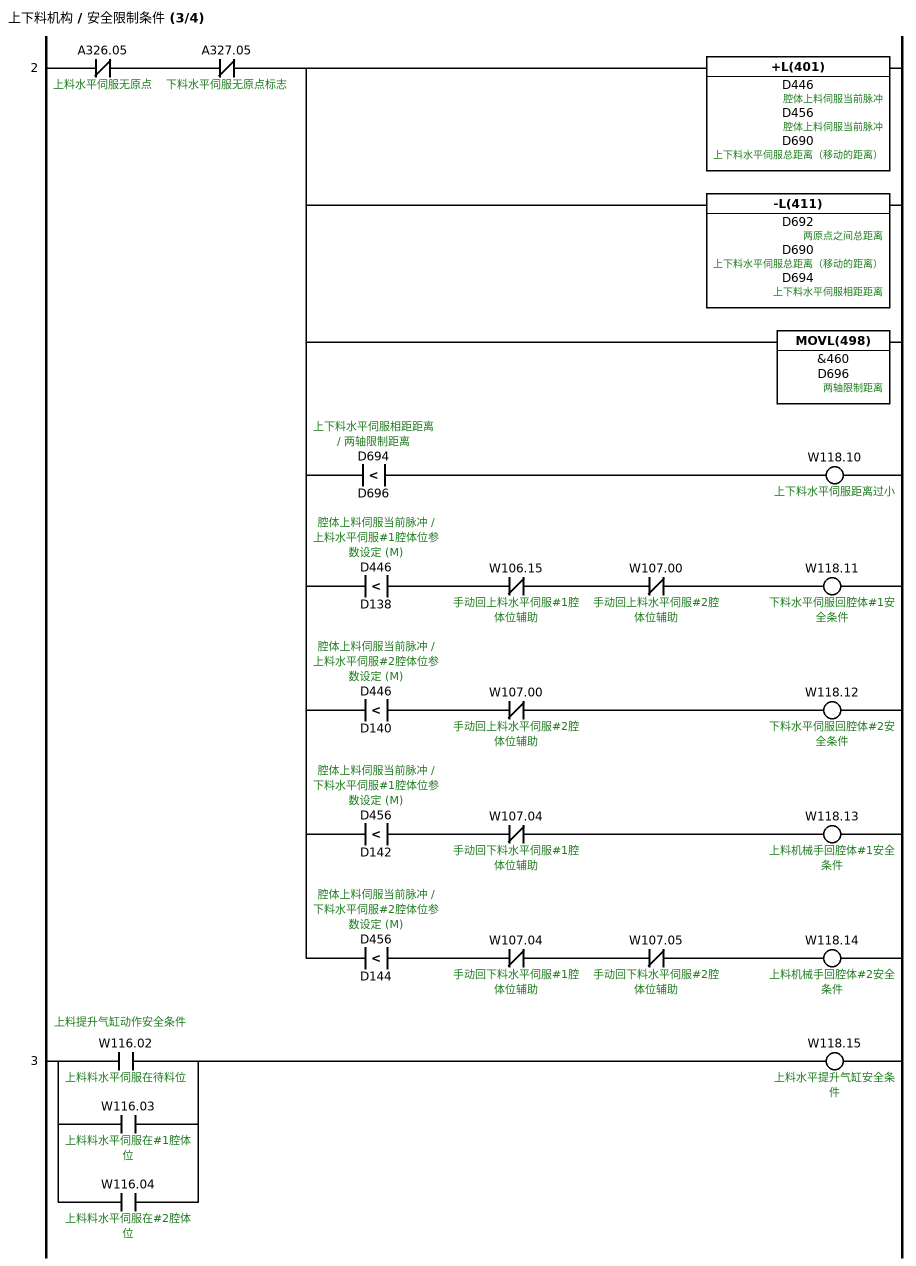
; rung 2
LDNOT A326.05  ; 上料水平伺服无原点
ANDNOT A327.05  ; 下料水平伺服无原点标志
OUT TR0
+L(401) D446 D456 D690  ; 腔体上料伺服当前脉冲, 上下料水平伺服总距离（移动的距离）
-L(411) D692 D690 D694  ; 两原点之间总距离, 上下料水平伺服总距离（移动的距离）, 上下料水平伺服相距距离
MOVL(498) &460 D696  ; 两轴限制距离
AND<L(311) D694 D696  ; 上下料水平伺服相距距离, 两轴限制距离
OUT W118.10  ; 上下料水平伺服距离过小
LD TR0
AND<L(311) D446 D138  ; 腔体上料伺服当前脉冲, 上料水平伺服#1腔体位参数设定 (M)
ANDNOT W106.15  ; 手动回上料水平伺服#1腔体位辅助
ANDNOT W107.00  ; 手动回上料水平伺服#2腔体位辅助
OUT W118.11  ; 下料水平伺服回腔体#1安全条件
LD TR0
AND<L(311) D446 D140  ; 腔体上料伺服当前脉冲, 上料水平伺服#2腔体位参数设定 (M)
ANDNOT W107.00  ; 手动回上料水平伺服#2腔体位辅助
OUT W118.12  ; 下料水平伺服回腔体#2安全条件
LD TR0
AND<L(311) D456 D142  ; 腔体上料伺服当前脉冲, 下料水平伺服#1腔体位参数设定 (M)
ANDNOT W107.04  ; 手动回下料水平伺服#1腔体位辅助
OUT W118.13  ; 上料机械手回腔体#1安全条件
LD TR0
AND<L(311) D456 D144  ; 腔体上料伺服当前脉冲, 下料水平伺服#2腔体位参数设定 (M)
ANDNOT W107.04  ; 手动回下料水平伺服#1腔体位辅助
ANDNOT W107.05  ; 手动回下料水平伺服#2腔体位辅助
OUT W118.14  ; 上料机械手回腔体#2安全条件
; rung 3: 上料提升气缸动作安全条件
LD W116.02  ; 上料料水平伺服在待料位
OR W116.03  ; 上料料水平伺服在#1腔体位
OR W116.04  ; 上料料水平伺服在#2腔体位
OUT W118.15  ; 上料水平提升气缸安全条件

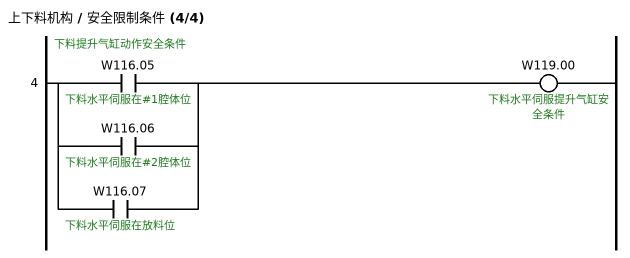
; rung 4: 下料提升气缸动作安全条件
LD W116.05  ; 下料水平伺服在#1腔体位
OR W116.06  ; 下料水平伺服在#2腔体位
OR W116.07  ; 下料水平伺服在放料位
OUT W119.00  ; 下料水平伺服提升气缸安全条件

### Section 上料、下料水平伺服参数设置

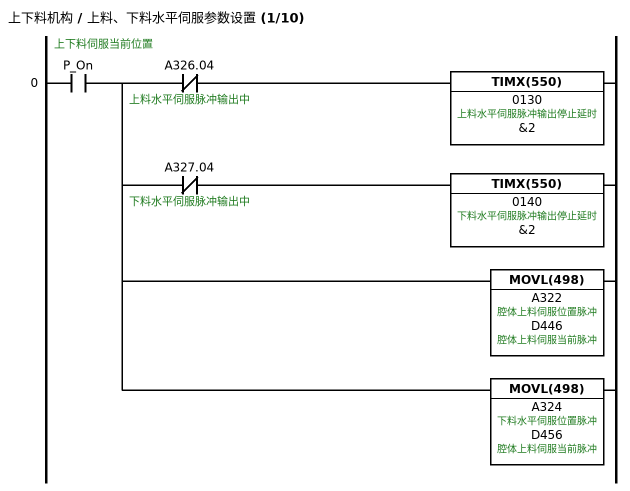
; rung 0: 上下料伺服当前位置
LD P_On
OUT TR0
ANDNOT A326.04  ; 上料水平伺服脉冲输出中
TIMX(550) 0130 &2  ; 上料水平伺服脉冲输出停止延时
LD TR0
ANDNOT A327.04  ; 下料水平伺服脉冲输出中
TIMX(550) 0140 &2  ; 下料水平伺服脉冲输出停止延时
LD TR0
MOVL(498) A322 D446  ; 腔体上料伺服位置脉冲, 腔体上料伺服当前脉冲
MOVL(498) A324 D456  ; 下料水平伺服位置脉冲, 腔体上料伺服当前脉冲

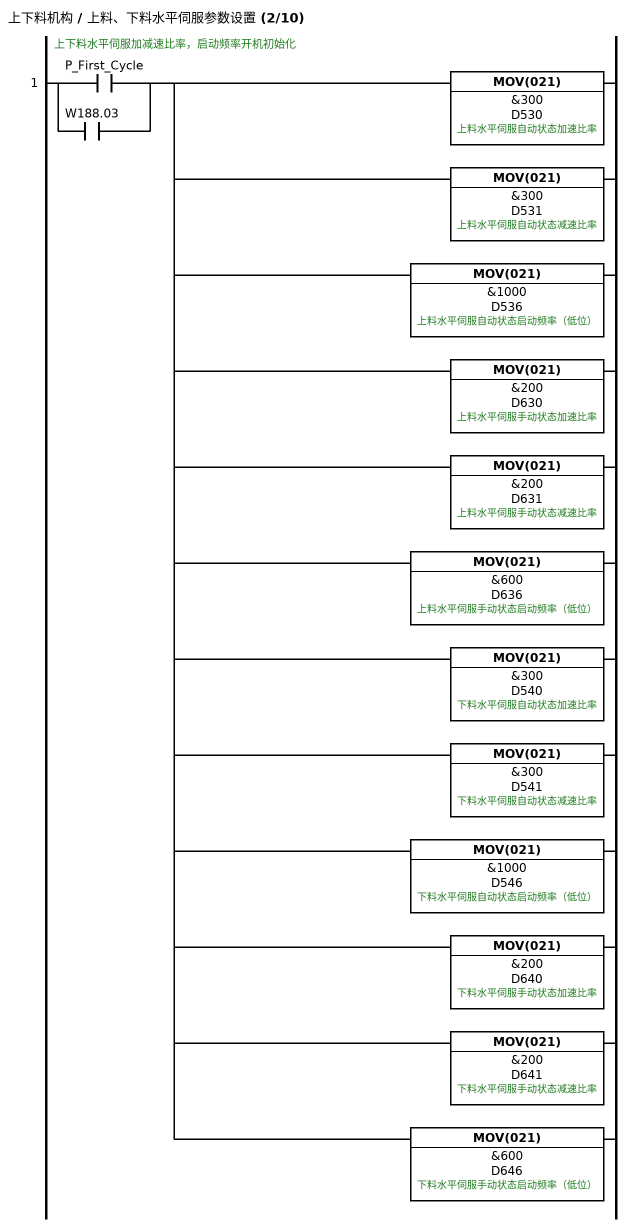
; rung 1: 上下料水平伺服加减速比率，启动频率开机初始化
LD P_First_Cycle
OR W188.03
MOV(021) &300 D530  ; 上料水平伺服自动状态加速比率
MOV(021) &300 D531  ; 上料水平伺服自动状态减速比率
MOV(021) &1000 D536  ; 上料水平伺服自动状态启动频率（低位）
MOV(021) &200 D630  ; 上料水平伺服手动状态加速比率
MOV(021) &200 D631  ; 上料水平伺服手动状态减速比率
MOV(021) &600 D636  ; 上料水平伺服手动状态启动频率（低位）
MOV(021) &300 D540  ; 下料水平伺服自动状态加速比率
MOV(021) &300 D541  ; 下料水平伺服自动状态减速比率
MOV(021) &1000 D546  ; 下料水平伺服自动状态启动频率（低位）
MOV(021) &200 D640  ; 下料水平伺服手动状态加速比率
MOV(021) &200 D641  ; 下料水平伺服手动状态减速比率
MOV(021) &600 D646  ; 下料水平伺服手动状态启动频率（低位）

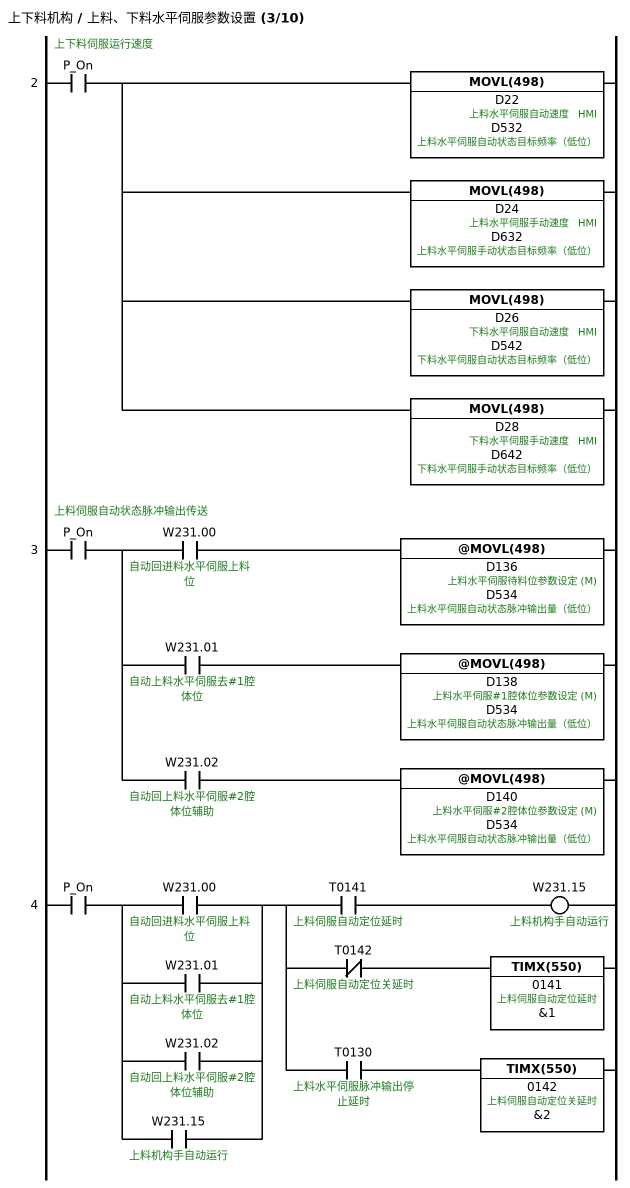
; rung 2: 上下料伺服运行速度
LD P_On
MOVL(498) D22 D532  ; 上料水平伺服自动速度   HMI, 上料水平伺服自动状态目标频率（低位）
MOVL(498) D24 D632  ; 上料水平伺服手动速度   HMI, 上料水平伺服手动状态目标频率（低位）
MOVL(498) D26 D542  ; 下料水平伺服自动速度   HMI, 下料水平伺服自动状态目标频率（低位）
MOVL(498) D28 D642  ; 下料水平伺服手动速度   HMI, 下料水平伺服手动状态目标频率（低位）
; rung 3: 上料伺服自动状态脉冲输出传送
LD P_On
OUT TR0
AND W231.00  ; 自动回进料水平伺服上料位
@MOVL(498) D136 D534  ; 上料水平伺服待料位参数设定 (M), 上料水平伺服自动状态脉冲输出量（低位）
LD TR0
AND W231.01  ; 自动上料水平伺服去#1腔体位
@MOVL(498) D138 D534  ; 上料水平伺服#1腔体位参数设定 (M), 上料水平伺服自动状态脉冲输出量（低位）
LD TR0
AND W231.02  ; 自动回上料水平伺服#2腔体位辅助
@MOVL(498) D140 D534  ; 上料水平伺服#2腔体位参数设定 (M), 上料水平伺服自动状态脉冲输出量（低位）
; rung 4
LD P_On
LD W231.00  ; 自动回进料水平伺服上料位
OR W231.01  ; 自动上料水平伺服去#1腔体位
OR W231.02  ; 自动回上料水平伺服#2腔体位辅助
OR W231.15  ; 上料机构手自动运行
ANDLD
OUT TR0
AND T0141  ; 上料伺服自动定位延时
OUT W231.15  ; 上料机构手自动运行
LD TR0
ANDNOT T0142  ; 上料伺服自动定位关延时
TIMX(550) 0141 &1  ; 上料伺服自动定位延时
LD TR0
AND T0130  ; 上料水平伺服脉冲输出停止延时
TIMX(550) 0142 &2  ; 上料伺服自动定位关延时

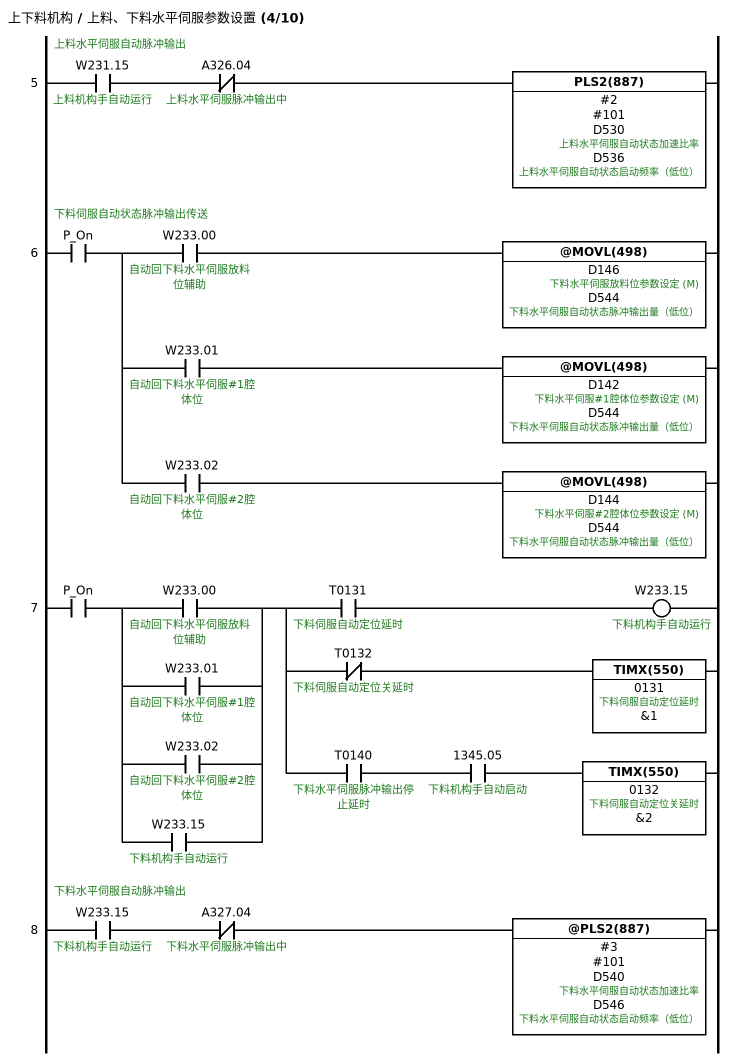
; rung 5: 上料水平伺服自动脉冲输出
LD W231.15  ; 上料机构手自动运行
ANDNOT A326.04  ; 上料水平伺服脉冲输出中
PLS2(887) #2 #101 D530 D536  ; 上料水平伺服自动状态加速比率, 上料水平伺服自动状态启动频率（低位）
; rung 6: 下料伺服自动状态脉冲输出传送
LD P_On
OUT TR0
AND W233.00  ; 自动回下料水平伺服放料位辅助
@MOVL(498) D146 D544  ; 下料水平伺服放料位参数设定 (M), 下料水平伺服自动状态脉冲输出量（低位）
LD TR0
AND W233.01  ; 自动回下料水平伺服#1腔体位
@MOVL(498) D142 D544  ; 下料水平伺服#1腔体位参数设定 (M), 下料水平伺服自动状态脉冲输出量（低位）
LD TR0
AND W233.02  ; 自动回下料水平伺服#2腔体位
@MOVL(498) D144 D544  ; 下料水平伺服#2腔体位参数设定 (M), 下料水平伺服自动状态脉冲输出量（低位）
; rung 7
LD P_On
LD W233.00  ; 自动回下料水平伺服放料位辅助
OR W233.01  ; 自动回下料水平伺服#1腔体位
OR W233.02  ; 自动回下料水平伺服#2腔体位
OR W233.15  ; 下料机构手自动运行
ANDLD
OUT TR0
AND T0131  ; 下料伺服自动定位延时
OUT W233.15  ; 下料机构手自动运行
LD TR0
ANDNOT T0132  ; 下料伺服自动定位关延时
TIMX(550) 0131 &1  ; 下料伺服自动定位延时
LD TR0
AND T0140  ; 下料水平伺服脉冲输出停止延时
AND 1345.05  ; 下料机构手自动启动
TIMX(550) 0132 &2  ; 下料伺服自动定位关延时
; rung 8: 下料水平伺服自动脉冲输出
LD W233.15  ; 下料机构手自动运行
ANDNOT A327.04  ; 下料水平伺服脉冲输出中
@PLS2(887) #3 #101 D540 D546  ; 下料水平伺服自动状态加速比率, 下料水平伺服自动状态启动频率（低位）

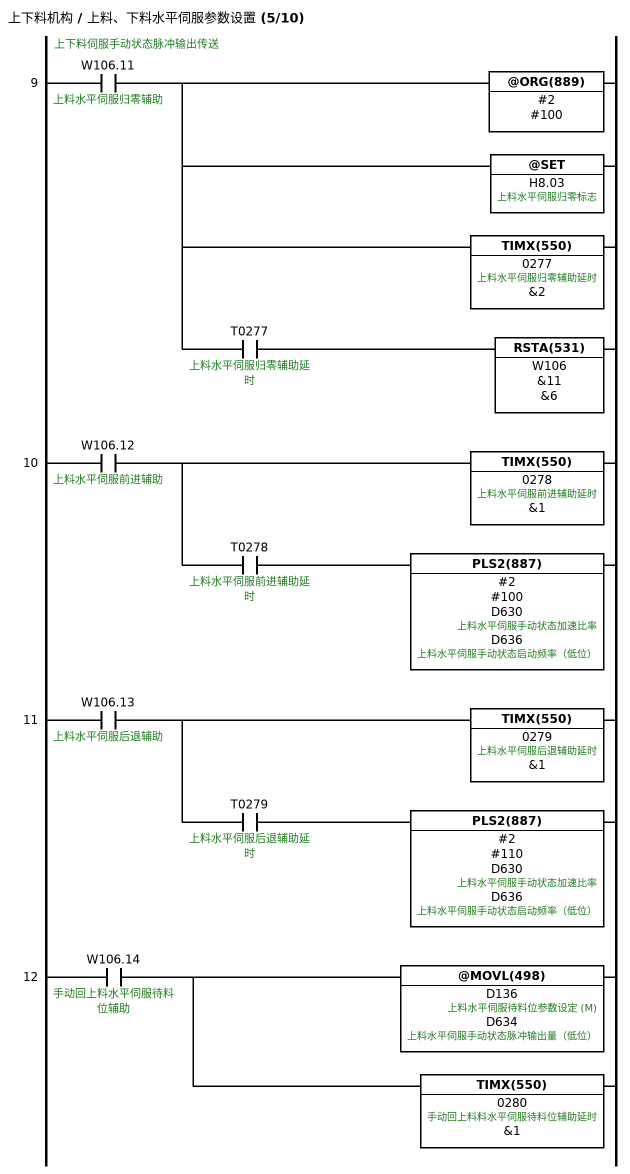
; rung 9: 上下料伺服手动状态脉冲输出传送
LD W106.11  ; 上料水平伺服归零辅助
@ORG(889) #2 #100
@SET H8.03  ; 上料水平伺服归零标志
TIMX(550) 0277 &2  ; 上料水平伺服归零辅助延时
AND T0277  ; 上料水平伺服归零辅助延时
RSTA(531) W106 &11 &6
; rung 10
LD W106.12  ; 上料水平伺服前进辅助
TIMX(550) 0278 &1  ; 上料水平伺服前进辅助延时
AND T0278  ; 上料水平伺服前进辅助延时
PLS2(887) #2 #100 D630 D636  ; 上料水平伺服手动状态加速比率, 上料水平伺服手动状态启动频率（低位）
; rung 11
LD W106.13  ; 上料水平伺服后退辅助
TIMX(550) 0279 &1  ; 上料水平伺服后退辅助延时
AND T0279  ; 上料水平伺服后退辅助延时
PLS2(887) #2 #110 D630 D636  ; 上料水平伺服手动状态加速比率, 上料水平伺服手动状态启动频率（低位）
; rung 12
LD W106.14  ; 手动回上料水平伺服待料位辅助
@MOVL(498) D136 D634  ; 上料水平伺服待料位参数设定 (M), 上料水平伺服手动状态脉冲输出量（低位）
TIMX(550) 0280 &1  ; 手动回上料料水平伺服待料位辅助延时

